FUNCTION_BLOCK COLOR_DECIDER (* Basic Function Block Type *)
  (* Standard: 61499-2 *)
  (* Version 0.3, 2009-09-15, JHC, Holobloc Inc, Changed transition priorities. *)
  (* Version 0.2, 2003-12-04, JHC, Rockwell Automation, Renamed for better indexing. *)
  (* Version 0.1, 2002-11-05, JHC, Rockwell Automation, Corrected missing ST element in Algorithm REQ. *)
  (* Version 0.0, 2000-05-30, JHC, Rockwell Automation *)
  PACKAGE fb.rt.Conveyer;
  IMPORT fb.datatype.*;
  IMPORT fb.rt.*;
  IMPORT fb.rt.mva.VSTYLE;
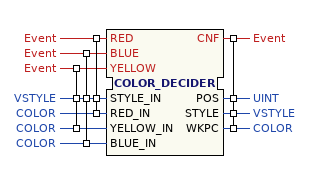
  EVENT_INPUT
    RED WITH STYLE_IN, RED_IN;
    BLUE WITH STYLE_IN, BLUE_IN;
    YELLOW WITH STYLE_IN, YELLOW_IN;
  END_EVENT
  EVENT_OUTPUT
    CNF WITH POS, STYLE, WKPC; (* Execution Confirmation *)
  END_EVENT
  VAR_INPUT
    STYLE_IN : VSTYLE;
    RED_IN : COLOR;
    YELLOW_IN : COLOR;
    BLUE_IN : COLOR;
  END_VAR
  VAR_OUTPUT
    POS : UINT := 0;
    STYLE : VSTYLE := PALLET;
    WKPC : COLOR;
  END_VAR
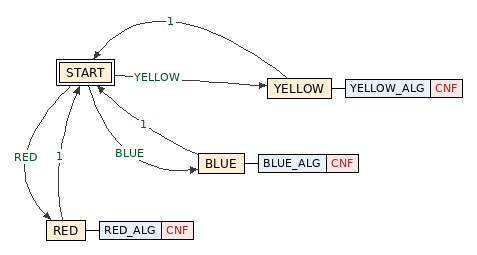
  EC_STATES
    START; (* Initial State *)
    RED : RED_ALG -> CNF;
    BLUE : BLUE_ALG -> CNF;
    YELLOW : YELLOW_ALG -> CNF;
  END_STATES
  EC_TRANSITIONS
    START TO RED := RED;
    RED TO START := 1;
    START TO BLUE := BLUE;
    BLUE TO START := 1;
    START TO YELLOW := YELLOW;
    YELLOW TO START := 1;
  END_TRANSITIONS
  ALGORITHM RED_ALG IN ST:
POS := 0;
STYLE := STYLE_IN;
WKPC := RED_IN;
  END_ALGORITHM
  ALGORITHM YELLOW_ALG IN ST:
POS := 0;
STYLE := STYLE_IN;
WKPC := YELLOW_IN;
  END_ALGORITHM
  ALGORITHM BLUE_ALG IN ST:
POS := 0;
STYLE := STYLE_IN;
WKPC := BLUE_IN;
  END_ALGORITHM
END_FUNCTION_BLOCK
